TYPE UBaseTypes_t :
UNION
	u8Value 	: USINT;
	s8Value 	: SINT;
	u16Value 	: UINT;
	s16Value 	: INT;
	u32Value 	: UDINT;
	s32Value 	: DINT;
	w16Value    : WORD;
	w32Value    : DWORD;
	r32Value 	: REAL;
	bValue		: BOOL;
END_UNION
END_TYPE

(* stored: Version 1.1.0.1, ProductVersion 3.1.4024.12
   DUT UBaseTypes_t: Id {2f74f94e-53a5-409d-a590-03080c2d19b5} *)
